SUBAPPLICATION Softkey_Aux_Button_IE (* Softkey_Aux_IE (SoftKey ODER AUX) ODER zusaetzlich ein weiterer Button (Button_IE, z.B. IO-Diag-Testbutton, kann aber auch ein regulaerer Button sein) aktiviert -> 1 gemeinsames IND-Event. Wie Softkey_Aux_Method_Button_IE, aber ohne die lokale OPC-UA-Methode - fuer Faelle, die nur SoftKey/AUX/Button gleichberechtigt brauchen. *)
  (* Standard: 61499-2; Description: Copyright (c) 2026 Meisterschulen am Ostbahnhof This program and the accompanying materials are made available under the terms of the Eclipse Public License 2.0 which is available at https://www.eclipse.org/legal/epl-2.0/ SPDX-License-Identifier: EPL-2.0 *)
  (* Version 1.0, 2026-09-15, Franz Höpfinger, Meisterschulen am Ostbahnhof, initial implementation - aus Baender_Individual_Toggle.SUB herausgeloest (dort 3x identisch fuer Igel/Elevator/Querband verdrahtet: Softkey_Aux_IE + Button_IE + E_MERGE_2). *)
  PACKAGE MyLib::sys;
  IMPORT isobus::UT::io::Button::ButtonActivationCode::BT_RELEASED_UNLATCHED;
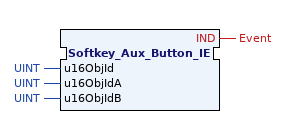
  EVENT_OUTPUT
    IND; (* Feuert wenn SoftKey, AUX ODER der Button aktiviert wird *)
  END_EVENT
  VAR_INPUT
    u16ObjId : UINT; (* Object ID SoftKey *)
    u16ObjIdA : UINT; (* Object ID AuxFunction2 *)
    u16ObjIdB : UINT; (* Object ID weiterer Button (z.B. IO-Diag-Testbutton), gleichberechtigt zu SoftKey/AUX *)
  END_VAR
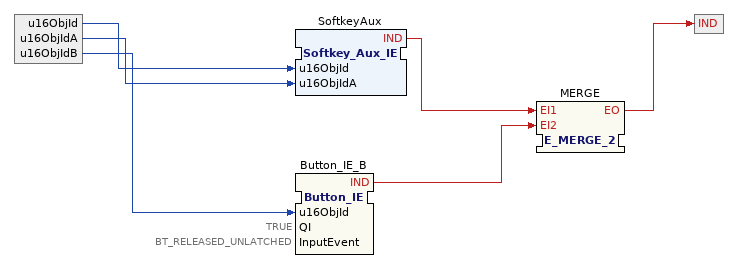
  FBS
    Button_IE_B : isobus::UT::io::Button::Button_IE(QI := TRUE, InputEvent := BT_RELEASED_UNLATCHED);
    MERGE : iec61499::events::E_MERGE_2;
  END_FBS
  SUBAPPS
    SoftkeyAux : MyLib::sys::Softkey_Aux_IE;
  END_SUBAPPS
  EVENT_CONNECTIONS
    SoftkeyAux.IND TO MERGE.EI1;
    Button_IE_B.IND TO MERGE.EI2;
    MERGE.EO TO IND;
  END_CONNECTIONS
  DATA_CONNECTIONS
    u16ObjId TO SoftkeyAux.u16ObjId;
    u16ObjIdA TO SoftkeyAux.u16ObjIdA;
    u16ObjIdB TO Button_IE_B.u16ObjId;
  END_CONNECTIONS
END_SUBAPPLICATION
